PROGRAM MAIN
VAR
END_VAR

END_PROGRAM

(* stored: Version 1.1.0.1
   POU MAIN: Id {8e3c4920-679f-48b6-bb0a-1f890bfb6a87} *)
